FUNCTION_BLOCK MOD_Crane
VAR_INPUT
	i_CraneDownSensor : MOD_Crane_I_stSensor;
	i_CraneUpSensor : MOD_Crane_I_stSensor;
	i_CraneAboveInput : MOD_Crane_I_stSensor;
	i_CraneAboveOutput : MOD_Crane_I_stSensor;

	i_Input : MOD_Crane_I_stLoad;
	i_LoadGrabbed : BOOL;
END_VAR
VAR_OUTPUT
	//right is down left is up
	q_HorizontalMotor : MOD_Crane_Q_stMotor;
	q_VerticalMotor : MOD_Crane_Q_stMotor;
	q_Grab : BOOL;
END_VAR
VAR_IN_OUT
	iq_CommandState : INT;
END_VAR
VAR
	State: INT := 10;
	MotorDirection : (Left, Right, Stopped);
	Executing : BOOL := FALSE;//variable for main state. used for orderly code		
END_VAR

CASE iq_CommandState OF
	Command.Error:
		Executing := FALSE;
		State := 10;//reset state
		q_VerticalMotor.MoveLeft := FALSE;
		q_VerticalMotor.MoveRight := FALSE;
		q_HorizontalMotor.MoveLeft := FALSE;
		q_HorizontalMotor.MoveRight := FALSE;
		
	Command.Executing:
		Executing := TRUE;
		
	Command.Pause:
		Executing := FALSE;
		q_VerticalMotor.MoveLeft := FALSE;
		q_VerticalMotor.MoveRight := FALSE;
		q_HorizontalMotor.MoveLeft := FALSE;
		q_HorizontalMotor.MoveRight := FALSE;
		
	Command.Reset:
		Executing := FALSE;
		State := 10;//reset state
		q_VerticalMotor.MoveLeft := FALSE;
		q_VerticalMotor.MoveRight := FALSE;
		q_HorizontalMotor.MoveLeft := FALSE;
		q_HorizontalMotor.MoveRight := FALSE;
		
	Command.Stop:
		Executing := FALSE;
		State := 10;//reset state
		q_VerticalMotor.MoveLeft := FALSE;
		q_VerticalMotor.MoveRight := FALSE;
		q_HorizontalMotor.MoveLeft := FALSE;
		q_HorizontalMotor.MoveRight := FALSE;	
		
END_CASE


IF Executing THEN
CASE State OF
	10://startup //reset?
		IF i_CraneAboveInput.Blocked THEN
			State := 20;
		ELSE
			State := 90;
		END_IF
		
	20://operational approval
		//wait untill
		IF i_Input.AllowedToOperate = TRUE THEN
			State := 21;
		END_IF
		
	21://check box ready
		//wait untill
		IF i_Input.Ready = TRUE THEN
			State := 30;
		END_IF
	
	30://move crane down
		
		q_VerticalMotor.MoveLeft := TRUE;
		q_VerticalMotor.MoveRight := FALSE;
		
		IF i_CraneDownSensor.Blocked = TRUE THEN
			State := 40;
		END_IF
		
	40://grab the load
		q_VerticalMotor.MoveLeft := FALSE;
		q_VerticalMotor.MoveRight := FALSE;
		q_HorizontalMotor.MoveLeft := FALSE;
		q_HorizontalMotor.MoveRight := FALSE;
		
		q_Grab := TRUE;
		
		IF i_LoadGrabbed = TRUE THEN
			State := 50;
		END_IF

	50://move crane up
		q_VerticalMotor.MoveLeft := TRUE;
		q_VerticalMotor.MoveRight := FALSE;
		q_HorizontalMotor.MoveLeft := FALSE;
		q_HorizontalMotor.MoveRight := FALSE;
		
		q_Grab := TRUE;
		
		IF i_CraneUpSensor.Blocked = TRUE THEN
			State := 60;
		END_IF

	60://move crane to output position
		q_VerticalMotor.MoveLeft := FALSE;
		q_VerticalMotor.MoveRight := FALSE;
		q_HorizontalMotor.MoveLeft := TRUE;
		q_HorizontalMotor.MoveRight := FALSE;
		
		q_Grab := TRUE;
		
		IF i_CraneAboveInput.Blocked = TRUE THEN
			State := 70;
		END_IF

	70://move crane down
		q_VerticalMotor.MoveLeft := FALSE;
		q_VerticalMotor.MoveRight := TRUE;
		q_HorizontalMotor.MoveLeft := FALSE;
		q_HorizontalMotor.MoveRight := FALSE;	
	
		IF i_CraneDownSensor.Blocked = TRUE THEN
			State := 80;
		END_IF

	80://release load
		q_Grab := FALSE;
		IF i_LoadGrabbed = FALSE THEN
			State := 90;
		END_IF

	90://move crane up
		q_VerticalMotor.MoveLeft := TRUE;
		q_VerticalMotor.MoveRight := FALSE;
		q_HorizontalMotor.MoveLeft := FALSE;
		q_HorizontalMotor.MoveRight := FALSE;	
		
		IF i_CraneUpSensor.Blocked = TRUE THEN
			State := 100;
		END_IF	

	100://move crane over input
		q_VerticalMotor.MoveLeft := FALSE;
		q_VerticalMotor.MoveRight := FALSE;
		q_HorizontalMotor.MoveLeft := FALSE;
		q_HorizontalMotor.MoveRight := TRUE;
			
		IF i_CraneAboveInput.Blocked = TRUE THEN
			State := 20;
		END_IF
END_CASE
END_IF

END_FUNCTION_BLOCK

(* stored: Version 1.1.0.1, ProductVersion 3.1.4024.6
   POU MOD_Crane: Id {5ef12530-d6be-413c-8970-2208adcc7e82}, SpecialFunc None *)
